(* This function block is different from the regular VRC in that CLOSING must be permitted. *)
FUNCTION_BLOCK FB_VRC_NO_FFO EXTENDS FB_VRC_NO
VAR_IN_OUT
    io_fbFFHWO    :    FB_HardwareFFOutput;
    fbArbiter: FB_Arbiter();
END_VAR
VAR_INPUT
    i_xPMPS_OK:	BOOL	; (*Set to True To switch off the bptm and PMPS Arbiter*)
    i_xIsAperture:BOOL :=FALSE; // Set tp True if this is an Aperture Valve, the MPS Fault will trip only when moving.
    i_sDevName : T_MaxString :=  'VRC_NO_FFO'; // Device name for diagnostic
    i_nTransitionRootID: UDINT; //A unique transition Root ID that is equal to or greater than 1000i_xIsAperture:BOOL :=FALSE; // Set tp True if this is an Aperture Valve, the MPS Fault will trip only when moving.
END_VAR
VAR_OUTPUT

END_VAR
VAR

    xPMPS_OK:	BOOL	; (*PMPS interlock*)
    bMoving : BOOL;
    bDone :BOOL;
    tBPTMtimeout:TON;
    bptm: BeamParameterTransitionManager;
    FFO    :    FB_FastFault :=(
        i_DevName := 'VRC_NO_FFO',
        i_Desc := 'Fault occurs when the valve is not in safe state',
        i_TypeCode := 16#1010);
    xMPS_OK:	BOOL; (*MPS Fast OK, is set when the Valve is Open*)

END_VAR

(*VRC_NO*)

(* This function block is different from the regular VRC in that CLOSING must be permitted. *)

(* On first PLC pass, put valve into vented state, which implies a closed valve *)
fbFSInit( CLK := TRUE, Q => xFirstPass);
IF xFirstPass THEN
    FFO.i_DevName := i_sDevName;
    iq_stValve.pv_xCLS_SW := FALSE;
	iq_stValve.eVGC_State := At_Vac;
END_IF




///Check valve position
IF iq_stValve.i_xClsLS AND  iq_stValve.i_xOpnLS THEN
    iq_stValve.eState:=INVALID;
ELSIF NOT iq_stValve.i_xClsLS AND iq_stValve.i_xOpnLS AND NOT iq_stValve.q_xCLS_DO THEN
    iq_stValve.eState:=OPEN;
ELSIF iq_stValve.i_xClsLS AND NOT iq_stValve.i_xOpnLS AND iq_stValve.q_xCLS_DO THEN
    iq_stValve.eState:=CLOSED;
ELSIF NOT iq_stValve.i_xClsLS AND NOT iq_stValve.i_xOpnLS THEN
    iq_stValve.eState:=MOVING;
ELSE
    iq_stValve.eState:=INVALID;
END_IF


(*evaluate Valve CLose external interlock*)
iq_stValve.xCLS_OK := i_xExtILK_OK;
IF NOT iq_stValve.xCLS_OK and NOT tonOvrd.Q THEN
    iq_stValve.pv_xCLS_SW := FALSE;
END_IF


(* Override logic *)
(* Goal: give ability to override, but do so in a way that people won't forget it.
Solution: Override only after ten seconds of override, protect against blips,
when the valve permission goes true for more than ten seconds consistently, remove override
*)

tonDelOK(IN:=iq_stValve.xCLS_OK, PT:=T#10S);
rtOK(CLK:=tonDelOK.Q);
IF rtOK.Q AND iq_stValve.pv_xOvrdCls THEN
    iq_stValve.pv_xOvrdCls :=FALSE;
    if (iq_stValve.eState=CLOSED) AND (i_xOverrideMode) THEN iq_stValve.pv_xCLS_SW := TRUE; END_IF
    //Log
    fbLogger(sMsg:='Override expired', eSevr:=TcEventSeverity.Warning);
END_IF

//Override timer
tonOvrd(IN:=iq_stValve.pv_xOvrdCls, PT:=tOvrd);

(* Here's where the valve Actuates *)
q_xCLS_DO := ((iq_stValve.xCLS_OK  AND iq_stValve.pv_xCLS_SW)OR (tonOvrd.Q AND i_xOverrideMode));
iq_stValve.q_xOPN_DO := NOT q_xCLS_DO;



///Check valve moving position timout
IF NOT iq_stValve.i_xClsLS AND tCLStimeout.Q THEN
    iq_stValve.bErrorPresent := TRUE;
    //iq_stValve.sErrorMessage := ' Close Timeout';
ELSIF NOT iq_stValve.i_xOpnLS AND tOPNtimeout.Q THEN
    iq_stValve.bErrorPresent := TRUE;
    //iq_stValve.sErrorMessage := ' Open Timeout';
END_IF
IF (iq_stValve.eState=INVALID) THEN
    iq_stValve.bErrorPresent := TRUE;
    //iq_stValve.sErrorMessage := CONCAT(sPath,' Invalid Valve Position');
END_IF

(*Timers*)
tOPNtimeout(IN:= NOT iq_stValve.q_xCLS_DO, PT := tTimeOutDuration );
tCLStimeout(IN:= iq_stValve.q_xCLS_DO, PT := tTimeOutDuration);


(*Soft IO Mapping*)
ACT_IO();

// Log States and triggers
ACT_Logger();




(*PMPS*)
IF NOT(i_xPMPS_OK) THEN
    ACT_PMPS();
END_IF
(*when interlock is lost the Valve closes regardless of the status of the PMPS and EPS*)
xPMPS_OK := i_xPMPS_OK OR (bptm.q_xTransitionAuthorized OR tBPTMtimeout.Q);
IF NOT (iq_stValve.xCLS_OK) THEN
    iq_stValve.pv_xCLS_SW:= FALSE; // Reset switch after inlk is lost
    iq_stValve.q_xCLS_DO := (iq_stValve.pv_xCLS_SW  AND iq_stValve.xCLS_OK) OR (tonOvrd.Q AND i_xOverrideMode);
ELSIF xPMPS_OK THEN
    iq_stValve.q_xCLS_DO := (iq_stValve.pv_xCLS_SW  AND iq_stValve.xCLS_OK) OR (tonOvrd.Q AND i_xOverrideMode);
//ELSIF NOT (i_xPMPS_OK) THEN
    // Only override mode
    //iq_stValve.q_xOPN_DO := (tonOvrd.Q AND i_xOverrideMode);
END_IF

(*MPS Fault setting*)
If (i_xIsAperture ) THEN
    (* When the valve  is open or in Closed position MPS is OK, Fault while moving*)
    xMPS_OK := (i_xOpnLS  AND NOT q_xCLS_DO) XOR (i_xClsLS  AND q_xCLS_DO);
ELSE
    (* When the valve  is open MPS is OK*)
    xMPS_OK := i_xOpnLS AND NOT i_xClsLS AND q_xCLS_DO;
END_IF

(*FAST FAULT*)
FFO(i_xOK := xMPS_OK,
    i_xReset := ,
    i_xAutoReset :=TRUE,
    io_fbFFHWO := io_fbFFHWO);

ACTION ACT_IO:
(*inputs*)
iq_stValve.i_xOpnLS := 	i_xOpnLS;
iq_stValve.i_xClsLS:=	i_xClsLS;
//iq_stValve. := i_xEXT_OK;
iq_stValve.xOverrideMode := i_xOverrideMode;
(*outputs*)
//q_xOPN_DO:= iq_stValve.q_xOPN_DO;
iq_stValve.q_xCLS_DO:= q_xCLS_DO;
END_ACTION

ACTION ACT_PMPS:
bMoving := (iq_stValve.pv_xCLS_SW AND NOT iq_stValve.i_xClsLS) XOR (NOT iq_stValve.pv_xCLS_SW AND NOT i_xOpnLS);
bDone := (NOT iq_stValve.pv_xCLS_SW AND iq_stValve.i_xOpnLS) XOR ( iq_stValve.pv_xCLS_SW AND i_xClsLS);
If (i_xIsAperture ) OR NOT (iq_stValve.pv_xCLS_SW )THEN
    bptm.i_stRequestedAssertion := PMPS_GVL.cstFullBeam;
ELSE  bptm.i_stRequestedAssertion := PMPS_GVL.cst0RateBeam;
END_IF
bptm(fbArbiter:=fbArbiter,
     i_TransitionAssertionID:=i_nTransitionRootID+2,
     i_stTransitionAssertion:=PMPS_GVL.cst0RateBeam,
     i_nRequestedAssertionID:=i_nTransitionRootID+ BOOL_TO_UDINT(NOT iq_stValve.pv_xCLS_SW),
     i_stRequestedAssertion:=,
     i_xMoving:=bMoving,
     i_xDoneMoving:= bDone,
     stCurrentBeamParameters:=PMPS_GVL.stCurrentBeamParameters,
     i_sDeviceName:=i_sDevName,
     q_xTransitionAuthorized=>);
// Timeout
tBPTMtimeout(IN:= bMoving AND NOT bptm.q_xTransitionAuthorized , PT:=T#1S);
//xPMPS_OK := bptm.q_xTransitionAuthorized OR tBPTMtimeout.Q;

//Timeout and clear request
IF (tBPTMtimeout.Q) THEN
    fbArbiter.RemoveRequest(bptm.i_TransitionAssertionID);
    fbArbiter.RemoveRequest(bptm.i_nRequestedAssertionID);
END_IF
END_ACTION

METHOD PUBLIC M_IsClosed : BOOL
VAR_INPUT
END_VAR
M_IsClosed := (This^.iq_stValve.eState = E_ValvePositionState.CLOSED);
END_METHOD

METHOD PUBLIC M_IsOpen : BOOL
VAR_INPUT
END_VAR
M_IsOpen := (This^.iq_stValve.eState = E_ValvePositionState.OPEN);
END_METHOD

// Use this Methode to Open or close the valve by setting the OPN_SW to the input value.
METHOD PUBLIC M_Set_CLS_SW : BOOL
VAR_INPUT
        value:BOOL;
END_VAR
This^.iq_stValve.pv_xCLS_SW := value;
END_METHOD

END_FUNCTION_BLOCK

(* stored: Version 1.1.0.1
   POU FB_VRC_NO_FFO: Id {c495bbea-0449-471b-ac8a-8e043f5385ad}, SpecialFunc None
   Action ACT_IO: Id {1d4a7f4f-4c3d-41ae-941b-94defd48f5cd}
   Action ACT_PMPS: Id {2d4909a8-c4a0-4b25-b483-8d410c71684c}
   Method M_IsClosed: Id {875acf97-80aa-44a2-9373-b2eb281de3fe}
   Method M_IsOpen: Id {4c54b83a-e3bf-491a-820f-87cfcefb4c61}
   Method M_Set_CLS_SW: Id {1fa8eeda-987c-48b9-9b68-226bece7fe9b} *)
